INTERFACE I_Station

METHOD ccl00_cycle : BOOL
VAR_INPUT
END_VAR
END_METHOD

METHOD ClearList : BOOL
VAR_INPUT
END_VAR
END_METHOD

PROPERTY InputConnections : I_Station
GET
END_GET
SET
END_SET
END_PROPERTY

PROPERTY OutputConnections : I_Station
GET
END_GET
SET
END_SET
END_PROPERTY

PROPERTY P_List : I_List
GET
END_GET
END_PROPERTY

PROPERTY P_List_Input_B : I_List
GET
END_GET
END_PROPERTY

PROPERTY P_List_Input_C : I_List
GET
END_GET
END_PROPERTY

PROPERTY P_nErrorCode : UDINT
GET
END_GET
END_PROPERTY

PROPERTY P_PositionOnTrack : ST_StationTrackPosition
GET
END_GET
END_PROPERTY

METHOD Processing : BOOL
VAR_INPUT
	i_nMachineState 	: INT;		// 1=Starting, 2=Running
END_VAR
END_METHOD

METHOD ResetStation : BOOL
VAR_INPUT
	bClear	: BOOL;
END_VAR
END_METHOD

END_INTERFACE

(* stored: Version 1.1.0.1, ProductVersion 3.1.4024.9
   Itf I_Station: Id {bca8b624-a113-4e00-aca3-b972bad40b56}
   Method ccl00_cycle: Id {a3d56f2d-b609-4967-9052-f42e09bd5bfc}
   Method ClearList: Id {d26a225f-ae2a-4d20-b875-2799e08aaf8f}
   Property InputConnections: Id {cdbffbd2-4001-44cf-bc5d-b6e772767b57}
   Get Get: Id {00ba5439-ccf4-4214-bed9-06a28b868650}
   Set Set: Id {34da8836-a7dc-49ad-b69d-ceb52d8eb184}
   Property OutputConnections: Id {dac74c09-a883-4cc2-bcee-9eff9898f6cc}
   Get Get: Id {14f3f06a-1e3b-4da0-8ae9-8be05da0f2a6}
   Set Set: Id {69a1e3a0-a154-4b4d-8815-bde5b641ee3b}
   Property P_List: Id {71df2070-bf2d-4865-ab6c-eac47b5aa035}
   Get Get: Id {3b58df1e-ed13-48d4-be1e-b54fa634e5e0}
   Property P_List_Input_B: Id {70373c47-8819-42ee-9d84-ed9f13a4226a}
   Get Get: Id {72457871-9bbe-401a-99ea-52c24c5246e3}
   Property P_List_Input_C: Id {3d333dfd-2088-49f9-9854-25ad6433250b}
   Get Get: Id {8e752642-c001-4ed8-90fc-4f1a78e6c835}
   Property P_nErrorCode: Id {adaa79df-fd38-47a9-8f02-41122f8130d9}
   Get Get: Id {d8ebd20d-6627-46e3-9009-d6c098e76fff}
   Property P_PositionOnTrack: Id {31956b21-1b46-440d-b828-c647302a1295}
   Get Get: Id {ed769a64-f884-4fca-a30b-27b6d292fa9f}
   Method Processing: Id {92f6ea25-c16c-402a-afde-b4604f3bd6de}
   Method ResetStation: Id {b1877d0f-e81a-48da-9418-04ae041b8a50} *)
